# EPICS IOC start-up script: require/3.1.2/siteMods/ipmiComm/4.2.0-rc.1/mtca3u_std.iocsh
#- ###   ESS MTCA Standard 3U Crate iocsh           ###
#- ####################################################
#- >> Mandatory
#- SESS           - SESSION NAME  (MUST BE lowercase)
#- INET           - IPMI SERVER INET
#- PREF           - PREFIX for the naming
#- >> Optional
#- PORT           - IPMI SERVER PORT, Default : 623
#- PROT           - IPMI SERVER PROTOCOL, Default : udp
#- PRIO           - PRIORITY
#- NOAUTOCONN     - Zero or missing indicates that portThread should automatically connect.
#- NOEOS          - asynInterposeEosConfig
#- LOCT           - Physical Location, Default : ""
#- ####################################################

drvAsynIPPortConfigure("$(SESS)","$(INET):$(PORT=623) $(PROT=udp)", $(PRIO=0), $(NOAUTOCONN=0), $(NOEOS=0))

mchInit("$(SESS)")

dbLoadRecords("mtca3u-crate-ess.db", "dev=$(PREF),link=$(SESS),location=$(LOCT=)")
